(* CoDeSys 2.3.9.55 project: pous.pro *)
(* Libraries: Standard.lib 2.6.14 11:37:46, IecSfc.lib 2.6.14 11:37:46, SYSLIBCALLBACK.LIB 2.6.14 12:06:08 *)

(* POU PLC_PRG, ST *)
PROGRAM PLC_PRG
VAR
	s1: BOOL;
	o2: BOOL;
END_VAR
s1:=o2;
END_PROGRAM
